TYPE csp_transfer_infeed_accumulation_belt_status_enum :(
	CSP_TRANSFER_INFEED_ACCUMULATION_BELT_STATUS_NOT_INITIALIZED 							:= 0,
	CSP_TRANSFER_INFEED_ACCUMULATION_BELT_STATUS_DISABLED 									:= 10,
	CSP_TRANSFER_INFEED_ACCUMULATION_BELT_STATUS_ENABLE_REQUEST 							:= 70,
	CSP_TRANSFER_INFEED_ACCUMULATION_BELT_STATUS_ENABLING 									:= 80,
	CSP_TRANSFER_INFEED_ACCUMULATION_BELT_STATUS_ENABLED 									:= 100,
	CSP_TRANSFER_INFEED_ACCUMULATION_BELT_STATUS_RUNNING									:= 110,
	CSP_TRANSFER_INFEED_ACCUMULATION_BELT_STATUS_STOP_REQUEST 								:= 500,
	CSP_TRANSFER_INFEED_ACCUMULATION_BELT_STATUS_DISABLE_REQUEST 							:= 530,
	CSP_TRANSFER_INFEED_ACCUMULATION_BELT_STATUS_DISABLING 									:= 540
	) := CSP_TRANSFER_INFEED_ACCUMULATION_BELT_STATUS_NOT_INITIALIZED;
END_TYPE

(* stored: Version 1.1.0.1, ProductVersion 3.1.4024.3
   DUT csp_transfer_infeed_accumulation_belt_status_enum: Id {6f86c232-2664-45c4-b1f6-82d3cb0fbb57} *)
